FUNCTION Convert_BYTE_TO_SINT : Hresult
VAR_INPUT
	in : BYTE;
	out : REFERENCE TO SINT;
END_VAR
VAR
	converted : SINT;
END_VAR

converted := BYTE_TO_SINT(in);

IF (SINT_TO_BYTE(converted) <> in) THEN
	Convert_BYTE_TO_SINT := INCOMPATIBLE;
	RETURN;
END_IF

out := converted;

END_FUNCTION

(* stored: Version 1.1.0.1, ProductVersion 3.1.4024.12
   POU Convert_BYTE_TO_SINT: Id {8eb20720-a6cd-4841-8b9b-6f5da59acd61}, SpecialFunc None *)
